FUNCTION_BLOCK AS2_TO_AS (* Composite FB for convert bidirectional AS2 to unidirectional AS *)
  (* Standard: 61499-2; Function: AS2_BIDIR forwards its incoming (EO1) side out as a plain unidirectional signal via AS_OUT. AS_IN publishes its value onto the outgoing (EI1) side of AS2_BIDIR.; Description: Copyright (c) 2026 HR Agrartechnik GmbH This program and the accompanying materials are made available under the terms of the Eclipse Public License 2.0 which is available at https://www.eclipse.org/legal/epl-2.0/ SPDX-License-Identifier: EPL-2.0 *)
  (* Version 1.0, 2026-09-12, Franz Höpfinger, HR Agrartechnik GmbH, Initial Version - Konvertierungsfamilie vervollstaendigt (analog zu AR2/AB2/AE2). *)
  PACKAGE adapter::conversion::bidirectional;
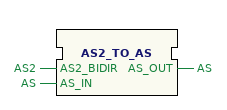
  SOCKETS
    AS2_BIDIR : adapter::types::bidirectional::AS2; (* Adapter Input: bidirectional tap, incoming side forwarded to AS_OUT, outgoing side driven by AS_IN *)
    AS_IN : adapter::types::unidirectional::AS; (* Adapter Input: unidirectional source *)
  END_SOCKETS
  PLUGS
    AS_OUT : adapter::types::unidirectional::AS; (* Adapter Output: mirrors AS2_BIDIR's incoming (indication) side *)
  END_PLUGS
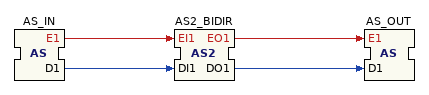
  EVENT_CONNECTIONS
    AS2_BIDIR.EO1 TO AS_OUT.E1;
    AS_IN.E1 TO AS2_BIDIR.EI1;
  END_CONNECTIONS
  DATA_CONNECTIONS
    AS2_BIDIR.DO1 TO AS_OUT.D1;
    AS_IN.D1 TO AS2_BIDIR.DI1;
  END_CONNECTIONS
END_FUNCTION_BLOCK
